ABB RAPID module: KennyTargets.mod

MODULE targets

	!Workplan Variables
	CONST string workplanName := "Kenny";
	CONST string workplanUUID := "4c150834-5da1-4e47-96b7-b16cde8d196c";

	!Workingsteps
	CONST string WorkPlan{20,6} := [
		["1","7", "Drilling.88", "5dba9a8c-05db-4595-a3ca-a7c776a922ef", "Hole.167", "f696efdc-798d-4b52-8da7-1cda0560be94"],
		["8","14", "Drilling.71", "36050cd1-dc9e-4879-8aed-1be84ca47fcc", "Hole.160", "7d9ff765-76db-4167-bb4c-53e49b398220"],
		["15","21", "Drilling.70", "4e2f8e6d-fe62-4a04-8e26-7213540deac3", "Hole.159", "eae91509-0626-466f-8bd8-d981c0f5cb83"],
		["22","28", "Drilling.87", "0659fa42-8109-4895-98a9-1d7bad19a7f8", "Hole.166", "d3306ec8-e7c0-4e48-ab13-ea87fff8c7f5"],
		["29","35", "Drilling.89", "25529f8b-f8c0-4dfe-8d3c-3ee9bb5aaf0b", "Hole.168", "45429ce3-7377-4a4c-ba7a-c1e998d11363"],
		["36","42", "Drilling.72", "0859f91d-f6a2-437f-b292-347030659a13", "Hole.161", "cfed41ef-af78-4deb-868f-e06b5c3e032d"],
		["43","49", "Drilling.87A", "bd213c16-608a-48e8-ba92-16dd103f0e82", "Hole.165", "e244bb89-273f-46de-9470-629b355579d0"],
		["50","56", "Drilling.72A", "30283c33-9bc4-4cb4-8bda-9191e9e1c1a8", "Hole.162", "6466e924-cde5-4cb9-be63-7b2e8a7ccfc9"],
		["57","63", "Drilling.51", "785224d9-9790-4c1a-a5a3-7fdee127c194", "Hole.149", "6ba27eaa-9f1f-4192-92ff-444f81e24c86"],
		["64","70", "Drilling.52", "6f0206cd-ac22-4230-a925-bd17b2c89fdf", "Hole.150", "7cbcafea-7ebf-4eb1-80bd-d38dc37e2ffa"],
		["71","77", "Drilling.52", "8223e776-d7de-4e22-b8f0-fb95f3561672", "Hole.151", "4113edcf-3075-48ef-82ea-78a646f36958"],
		["78","84", "Drilling.53", "15048da7-3430-4dce-a3f8-5c07c276276c", "Hole.152", "8d763157-3777-4192-8350-24f7dbecc6a9"],
		["85","91", "Drilling.66", "95c1f94a-95c9-4216-a369-009bc624fa7c", "Hole.155", "7352fd5f-6f0d-4d28-bb2c-b9767f2ea8ca"],
		["92","98", "Drilling.67", "f632f581-ae96-402c-b4f7-e3bd5086856f", "Hole.156", "7c20ef06-77fc-43ec-8049-9df34a187736"],
		["99","105", "Drilling.68", "c8ae3b54-663b-4d09-baf6-4b0ee80be638", "Hole.157", "0e7d8ffe-7fd5-4dd5-9f70-b0b78f8877dc"],
		["106","112", "Drilling.69", "d220337c-e0a3-4693-a211-54c62b6cd64b", "Hole.158", "6fcc203b-750e-4cab-906d-26d0a8242386"],
		["113","119", "Drilling.90", "f0f7cb38-96f5-48d3-840e-edf378bb551b", "Hole.170", "636bd456-6d68-43b2-b22b-21d689faa8d2"],
		["120","126", "Drilling.91", "abcac725-976e-4a50-a32b-3dd65c42f522", "Hole.171", "d8ca9eb0-5b5f-4eba-8f6d-b2fe1a9acaf1"],
		["127","133", "Drilling.92", "0d36731a-94ab-4213-8ec9-dfebb0effafd", "Hole.172", "f87e6c87-82b4-4795-8769-a91132110e61"],
		["134","140", "Drilling.93", "7777f709-fc7f-49f0-a947-dc19bdc87d5a", "Hole.173", "76d0f419-d37b-4108-8258-5a43c85176e2"]
		];

	!Positions
	CONST robtarget WorkingstepRobtargets{140} := [
		[[1251.36031479439,159.986015149395,27.4616252468863],[0.00827389312568621,0.000714793553765205,-0.996254662433507,0.0860678763663786],[0,0,0,0],[9E+09,9E+09,9E+09,9E+09,9E+09,9E+09]],
		[[1250.52908619628,151.273669125687,-22.5787992695068],[0.00827389312568621,0.000714793553765205,-0.996254662433507,0.0860678763663786],[0,0,0,0],[9E+09,9E+09,9E+09,9E+09,9E+09,9E+09]],
		[[1250.52908619628,151.273669125687,-22.5787992695068],[0.00827389312568621,0.000714793553765205,-0.996254662433507,0.0860678763663786],[0,0,0,0],[9E+09,9E+09,9E+09,9E+09,9E+09,9E+09]],
		[[1250.00956832245,145.828452860869,-53.8540645922525],[0.00827389312568621,0.000714793553765205,-0.996254662433507,0.0860678763663786],[0,0,0,0],[9E+09,9E+09,9E+09,9E+09,9E+09,9E+09]],
		[[1250.00956832245,145.828452860869,-53.8540645922525],[0.00827389312568621,0.000714793553765205,-0.996254662433507,0.0860678763663786],[0,0,0,0],[9E+09,9E+09,9E+09,9E+09,9E+09,9E+09]],
		[[1250.52908619628,151.273669125687,-22.5787992695068],[0.00827389312568621,0.000714793553765205,-0.996254662433507,0.0860678763663786],[0,0,0,0],[9E+09,9E+09,9E+09,9E+09,9E+09,9E+09]],
		[[1251.36031479439,159.986015149395,27.4616252468863],[0.00827389312568621,0.000714793553765205,-0.996254662433507,0.0860678763663786],[0,0,0,0],[9E+09,9E+09,9E+09,9E+09,9E+09,9E+09]],
		[[1190.56655432575,165.147556673713,27.5696380197376],[0.00833481880816476,0.000730999019406425,-0.996141160359995,0.0873658118059379],[0,0,0,0],[9E+09,9E+09,9E+09,9E+09,9E+09,9E+09]],
		[[1189.72949308332,156.304823646231,-22.4478129457116],[0.00833481880816476,0.000730999019406425,-0.996141160359995,0.0873658118059379],[0,0,0,0],[9E+09,9E+09,9E+09,9E+09,9E+09,9E+09]],
		[[1189.72949308332,156.304823646231,-22.4478129457116],[0.00833481880816476,0.000730999019406425,-0.996141160359995,0.0873658118059379],[0,0,0,0],[9E+09,9E+09,9E+09,9E+09,9E+09,9E+09]],
		[[1189.2063298068,150.778115504055,-53.7087197991172],[0.00833481880816476,0.000730999019406425,-0.996141160359995,0.0873658118059379],[0,0,0,0],[9E+09,9E+09,9E+09,9E+09,9E+09,9E+09]],
		[[1189.2063298068,150.778115504055,-53.7087197991172],[0.00833481880816476,0.000730999019406425,-0.996141160359995,0.0873658118059379],[0,0,0,0],[9E+09,9E+09,9E+09,9E+09,9E+09,9E+09]],
		[[1189.72949308332,156.304823646231,-22.4478129457116],[0.00833481880816476,0.000730999019406425,-0.996141160359995,0.0873658118059379],[0,0,0,0],[9E+09,9E+09,9E+09,9E+09,9E+09,9E+09]],
		[[1190.56655432575,165.147556673713,27.5696380197376],[0.00833481880816476,0.000730999019406425,-0.996141160359995,0.0873658118059379],[0,0,0,0],[9E+09,9E+09,9E+09,9E+09,9E+09,9E+09]],
		[[1191.89415560584,213.973804453541,17.5823830985576],[0.00973585929847244,0.00111256490306083,-0.993486175232847,0.113530589993472],[0,0,0,0],[9E+09,9E+09,9E+09,9E+09,9E+09,9E+09]],
		[[1190.92426864878,202.513131068111,-31.8984443484752],[0.00973585929847244,0.00111256490306083,-0.993486175232847,0.113530589993472],[0,0,0,0],[9E+09,9E+09,9E+09,9E+09,9E+09,9E+09]],
		[[1190.92426864878,202.513131068111,-31.8984443484752],[0.00973585929847244,0.00111256490306083,-0.993486175232847,0.113530589993472],[0,0,0,0],[9E+09,9E+09,9E+09,9E+09,9E+09,9E+09]],
		[[1190.31808930061,195.350210202218,-62.8239615028704],[0.00973585929847244,0.00111256490306083,-0.993486175232847,0.113530589993472],[0,0,0,0],[9E+09,9E+09,9E+09,9E+09,9E+09,9E+09]],
		[[1190.31808930061,195.350210202218,-62.8239615028704],[0.00973585929847244,0.00111256490306083,-0.993486175232847,0.113530589993472],[0,0,0,0],[9E+09,9E+09,9E+09,9E+09,9E+09,9E+09]],
		[[1190.92426864878,202.513131068111,-31.8984443484752],[0.00973585929847244,0.00111256490306083,-0.993486175232847,0.113530589993472],[0,0,0,0],[9E+09,9E+09,9E+09,9E+09,9E+09,9E+09]],
		[[1191.89415560584,213.973804453541,17.5823830985576],[0.00973585929847244,0.00111256490306083,-0.993486175232847,0.113530589993472],[0,0,0,0],[9E+09,9E+09,9E+09,9E+09,9E+09,9E+09]],
		[[1251.50868656169,112.759337427171,34.4420178830909],[0.00729205985071979,0.000442363584144468,-0.998138382466358,0.0605508020180991],[0,0,0,0],[9E+09,9E+09,9E+09,9E+09,9E+09,9E+09]],
		[[1250.77191390728,106.618500806138,-15.9800734226999],[0.00729205985071979,0.000442363584144468,-0.998138382466358,0.0605508020180991],[0,0,0,0],[9E+09,9E+09,9E+09,9E+09,9E+09,9E+09]],
		[[1250.77191390728,106.618500806138,-15.9800734226999],[0.00729205985071979,0.000442363584144468,-0.998138382466358,0.0605508020180991],[0,0,0,0],[9E+09,9E+09,9E+09,9E+09,9E+09,9E+09]],
		[[1250.31143099827,102.780477917993,-47.4938804888192],[0.00729205985071979,0.000442363584144468,-0.998138382466358,0.0605508020180991],[0,0,0,0],[9E+09,9E+09,9E+09,9E+09,9E+09,9E+09]],
		[[1250.31143099827,102.780477917993,-47.4938804888192],[0.00729205985071979,0.000442363584144468,-0.998138382466358,0.0605508020180991],[0,0,0,0],[9E+09,9E+09,9E+09,9E+09,9E+09,9E+09]],
		[[1250.77191390728,106.618500806138,-15.9800734226999],[0.00729205985071979,0.000442363584144468,-0.998138382466358,0.0605508020180991],[0,0,0,0],[9E+09,9E+09,9E+09,9E+09,9E+09,9E+09]],
		[[1251.50868656169,112.759337427171,34.4420178830909],[0.00729205985071979,0.000442363584144468,-0.998138382466358,0.0605508020180991],[0,0,0,0],[9E+09,9E+09,9E+09,9E+09,9E+09,9E+09]],
		[[1251.8601825108,210.524561887497,17.2060251950538],[0.0097362625680173,0.00111307904909481,-0.993480782143631,0.113577734426767],[0,0,0,0],[9E+09,9E+09,9E+09,9E+09,9E+09,9E+09]],
		[[1250.89027144533,199.059191507408,-32.2737136338089],[0.0097362625680173,0.00111307904909481,-0.993480782143631,0.113577734426767],[0,0,0,0],[9E+09,9E+09,9E+09,9E+09,9E+09,9E+09]],
		[[1250.89027144533,199.059191507408,-32.2737136338089],[0.0097362625680173,0.00111307904909481,-0.993480782143631,0.113577734426767],[0,0,0,0],[9E+09,9E+09,9E+09,9E+09,9E+09,9E+09]],
		[[1250.28407702942,191.893335019853,-63.1985504018481],[0.0097362625680173,0.00111307904909481,-0.993480782143631,0.113577734426767],[0,0,0,0],[9E+09,9E+09,9E+09,9E+09,9E+09,9E+09]],
		[[1250.28407702942,191.893335019853,-63.1985504018481],[0.0097362625680173,0.00111307904909481,-0.993480782143631,0.113577734426767],[0,0,0,0],[9E+09,9E+09,9E+09,9E+09,9E+09,9E+09]],
		[[1250.89027144533,199.059191507408,-32.2737136338089],[0.0097362625680173,0.00111307904909481,-0.993480782143631,0.113577734426767],[0,0,0,0],[9E+09,9E+09,9E+09,9E+09,9E+09,9E+09]],
		[[1251.8601825108,210.524561887497,17.2060251950538],[0.0097362625680173,0.00111307904909481,-0.993480782143631,0.113577734426767],[0,0,0,0],[9E+09,9E+09,9E+09,9E+09,9E+09,9E+09]],
		[[1190.88023867958,116.257500079554,34.9005826267419],[0.00731948636979851,0.000450203628618277,-0.998086922900926,0.0613898751435108],[0,0,0,0],[9E+09,9E+09,9E+09,9E+09,9E+09,9E+09]],
		[[1190.14080955814,110.031886232754,-15.5110725415314],[0.00731948636979851,0.000450203628618277,-0.998086922900926,0.0613898751435108],[0,0,0,0],[9E+09,9E+09,9E+09,9E+09,9E+09,9E+09]],
		[[1190.14080955814,110.031886232754,-15.5110725415314],[0.00731948636979851,0.000450203628618277,-0.998086922900926,0.0613898751435108],[0,0,0,0],[9E+09,9E+09,9E+09,9E+09,9E+09,9E+09]],
		[[1189.67866635724,106.140877578504,-47.0183570217021],[0.00731948636979851,0.000450203628618277,-0.998086922900926,0.0613898751435108],[0,0,0,0],[9E+09,9E+09,9E+09,9E+09,9E+09,9E+09]],
		[[1189.67866635724,106.140877578504,-47.0183570217021],[0.00731948636979851,0.000450203628618277,-0.998086922900926,0.0613898751435108],[0,0,0,0],[9E+09,9E+09,9E+09,9E+09,9E+09,9E+09]],
		[[1190.14080955814,110.031886232754,-15.5110725415314],[0.00731948636979851,0.000450203628618277,-0.998086922900926,0.0613898751435108],[0,0,0,0],[9E+09,9E+09,9E+09,9E+09,9E+09,9E+09]],
		[[1190.88023867958,116.257500079554,34.9005826267419],[0.00731948636979851,0.000450203628618277,-0.998086922900926,0.0613898751435108],[0,0,0,0],[9E+09,9E+09,9E+09,9E+09,9E+09,9E+09]],
		[[1250.76447640153,68.6402546108708,38.7643104755585],[0.00669120018047459,0.000246507461145111,-0.999299675598547,0.0368147446392719],[0,0,0,0],[9E+09,9E+09,9E+09,9E+09,9E+09,9E+09]],
		[[1250.08604859299,64.9023284513774,-11.8934396100383],[0.00669120018047459,0.000246507461145111,-0.999299675598547,0.0368147446392719],[0,0,0,0],[9E+09,9E+09,9E+09,9E+09,9E+09,9E+09]],
		[[1250.08604859299,64.9023284513774,-11.8934396100383],[0.00669120018047459,0.000246507461145111,-0.999299675598547,0.0368147446392719],[0,0,0,0],[9E+09,9E+09,9E+09,9E+09,9E+09,9E+09]],
		[[1249.66203121265,62.5661246016938,-43.5545334135362],[0.00669120018047459,0.000246507461145111,-0.999299675598547,0.0368147446392719],[0,0,0,0],[9E+09,9E+09,9E+09,9E+09,9E+09,9E+09]],
		[[1249.66203121265,62.5661246016938,-43.5545334135362],[0.00669120018047459,0.000246507461145111,-0.999299675598547,0.0368147446392719],[0,0,0,0],[9E+09,9E+09,9E+09,9E+09,9E+09,9E+09]],
		[[1250.08604859299,64.9023284513774,-11.8934396100383],[0.00669120018047459,0.000246507461145111,-0.999299675598547,0.0368147446392719],[0,0,0,0],[9E+09,9E+09,9E+09,9E+09,9E+09,9E+09]],
		[[1250.76447640153,68.6402546108708,38.7643104755585],[0.00669120018047459,0.000246507461145111,-0.999299675598547,0.0368147446392719],[0,0,0,0],[9E+09,9E+09,9E+09,9E+09,9E+09,9E+09]],
		[[1189.9772715838,69.4582698852428,39.5179868929106],[0.00668793620390687,0.000245146305514718,-0.999306502156587,0.0366295803987568],[0,0,0,0],[9E+09,9E+09,9E+09,9E+09,9E+09,9E+09]],
		[[1189.29916082133,65.7391188387643,-11.1411493145624],[0.00668793620390687,0.000245146305514718,-0.999306502156587,0.0366295803987568],[0,0,0,0],[9E+09,9E+09,9E+09,9E+09,9E+09,9E+09]],
		[[1189.29916082133,65.7391188387643,-11.1411493145624],[0.00668793620390687,0.000245146305514718,-0.999306502156587,0.0366295803987568],[0,0,0,0],[9E+09,9E+09,9E+09,9E+09,9E+09,9E+09]],
		[[1188.87534159478,63.4146494347152,-42.803109444233],[0.00668793620390687,0.000245146305514718,-0.999306502156587,0.0366295803987568],[0,0,0,0],[9E+09,9E+09,9E+09,9E+09,9E+09,9E+09]],
		[[1188.87534159478,63.4146494347152,-42.803109444233],[0.00668793620390687,0.000245146305514718,-0.999306502156587,0.0366295803987568],[0,0,0,0],[9E+09,9E+09,9E+09,9E+09,9E+09,9E+09]],
		[[1189.29916082133,65.7391188387643,-11.1411493145624],[0.00668793620390687,0.000245146305514718,-0.999306502156587,0.0366295803987568],[0,0,0,0],[9E+09,9E+09,9E+09,9E+09,9E+09,9E+09]],
		[[1189.9772715838,69.4582698852428,39.5179868929106],[0.00668793620390687,0.000245146305514718,-0.999306502156587,0.0366295803987568],[0,0,0,0],[9E+09,9E+09,9E+09,9E+09,9E+09,9E+09]],
		[[1048.75377702369,221.064248736861,18.7456359573398],[0.00969862451718228,0.0011013674490227,-0.993566525165611,0.112828559073272],[0,0,0,0],[9E+09,9E+09,9E+09,9E+09,9E+09,9E+09]],
		[[1047.78736158715,209.673531246336,-30.7514103813565],[0.00969862451718228,0.0011013674490227,-0.993566525165611,0.112828559073272],[0,0,0,0],[9E+09,9E+09,9E+09,9E+09,9E+09,9E+09]],
		[[1047.78736158715,209.673531246336,-30.7514103813565],[0.00969862451718228,0.0011013674490227,-0.993566525165611,0.112828559073272],[0,0,0,0],[9E+09,9E+09,9E+09,9E+09,9E+09,9E+09]],
		[[1047.18335193931,202.554332814758,-61.6870643430416],[0.00969862451718228,0.0011013674490227,-0.993566525165611,0.112828559073272],[0,0,0,0],[9E+09,9E+09,9E+09,9E+09,9E+09,9E+09]],
		[[1047.18335193931,202.554332814758,-61.6870643430416],[0.00969862451718228,0.0011013674490227,-0.993566525165611,0.112828559073272],[0,0,0,0],[9E+09,9E+09,9E+09,9E+09,9E+09,9E+09]],
		[[1047.78736158715,209.673531246336,-30.7514103813565],[0.00969862451718228,0.0011013674490227,-0.993566525165611,0.112828559073272],[0,0,0,0],[9E+09,9E+09,9E+09,9E+09,9E+09,9E+09]],
		[[1048.75377702369,221.064248736861,18.7456359573398],[0.00969862451718228,0.0011013674490227,-0.993566525165611,0.112828559073272],[0,0,0,0],[9E+09,9E+09,9E+09,9E+09,9E+09,9E+09]],
		[[1049.72266482233,161.388258470636,30.5369306758237],[0.00810433453815839,0.000668070226723706,-0.996586609691307,0.0821523148051996],[0,0,0,0],[9E+09,9E+09,9E+09,9E+09,9E+09,9E+09]],
		[[1048.90765118534,153.069523657326,-19.5706975246546],[0.00810433453815839,0.000668070226723706,-0.996586609691307,0.0821523148051996],[0,0,0,0],[9E+09,9E+09,9E+09,9E+09,9E+09,9E+09]],
		[[1048.90765118534,153.069523657326,-19.5706975246546],[0.00810433453815839,0.000668070226723706,-0.996586609691307,0.0821523148051996],[0,0,0,0],[9E+09,9E+09,9E+09,9E+09,9E+09,9E+09]],
		[[1048.39826766222,147.870314399008,-50.8879651499535],[0.00810433453815839,0.000668070226723706,-0.996586609691307,0.0821523148051996],[0,0,0,0],[9E+09,9E+09,9E+09,9E+09,9E+09,9E+09]],
		[[1048.39826766222,147.870314399008,-50.8879651499535],[0.00810433453815839,0.000668070226723706,-0.996586609691307,0.0821523148051996],[0,0,0,0],[9E+09,9E+09,9E+09,9E+09,9E+09,9E+09]],
		[[1048.90765118534,153.069523657326,-19.5706975246546],[0.00810433453815839,0.000668070226723706,-0.996586609691307,0.0821523148051996],[0,0,0,0],[9E+09,9E+09,9E+09,9E+09,9E+09,9E+09]],
		[[1049.72266482233,161.388258470636,30.5369306758237],[0.00810433453815839,0.000668070226723706,-0.996586609691307,0.0821523148051996],[0,0,0,0],[9E+09,9E+09,9E+09,9E+09,9E+09,9E+09]],
		[[1050.01208432635,107.933890240474,37.9095374224083],[0.007122245347503,0.00039121136422263,-0.998469455496607,0.0548440244255241],[0,0,0,0],[9E+09,9E+09,9E+09,9E+09,9E+09,9E+09]],
		[[1049.29175162139,102.369982698389,-12.5797094887637],[0.007122245347503,0.00039121136422263,-0.998469455496607,0.0548440244255241],[0,0,0,0],[9E+09,9E+09,9E+09,9E+09,9E+09,9E+09]],
		[[1049.29175162139,102.369982698389,-12.5797094887637],[0.007122245347503,0.00039121136422263,-0.998469455496607,0.0548440244255241],[0,0,0,0],[9E+09,9E+09,9E+09,9E+09,9E+09,9E+09]],
		[[1048.84154368078,98.8925404845857,-44.1354888082459],[0.007122245347503,0.00039121136422263,-0.998469455496607,0.0548440244255241],[0,0,0,0],[9E+09,9E+09,9E+09,9E+09,9E+09,9E+09]],
		[[1048.84154368078,98.8925404845857,-44.1354888082459],[0.007122245347503,0.00039121136422263,-0.998469455496607,0.0548440244255241],[0,0,0,0],[9E+09,9E+09,9E+09,9E+09,9E+09,9E+09]],
		[[1049.29175162139,102.369982698389,-12.5797094887637],[0.007122245347503,0.00039121136422263,-0.998469455496607,0.0548440244255241],[0,0,0,0],[9E+09,9E+09,9E+09,9E+09,9E+09,9E+09]],
		[[1050.01208432635,107.933890240474,37.9095374224083],[0.007122245347503,0.00039121136422263,-0.998469455496607,0.0548440244255241],[0,0,0,0],[9E+09,9E+09,9E+09,9E+09,9E+09,9E+09]],
		[[1048.45280482734,61.188425000286,41.9579660547863],[0.00659046299640987,0.00020471594525679,-0.999496183042603,0.0310468029294715],[0,0,0,0],[9E+09,9E+09,9E+09,9E+09,9E+09,9E+09]],
		[[1047.78419688503,58.0355219643173,-8.73968838666952],[0.00659046299640987,0.00020471594525679,-0.999496183042603,0.0310468029294715],[0,0,0,0],[9E+09,9E+09,9E+09,9E+09,9E+09,9E+09]],
		[[1047.78419688503,58.0355219643173,-8.73968838666952],[0.00659046299640987,0.00020471594525679,-0.999496183042603,0.0310468029294715],[0,0,0,0],[9E+09,9E+09,9E+09,9E+09,9E+09,9E+09]],
		[[1047.36631692108,56.064957566837,-40.4257224125791],[0.00659046299640987,0.00020471594525679,-0.999496183042603,0.0310468029294715],[0,0,0,0],[9E+09,9E+09,9E+09,9E+09,9E+09,9E+09]],
		[[1047.36631692108,56.064957566837,-40.4257224125791],[0.00659046299640987,0.00020471594525679,-0.999496183042603,0.0310468029294715],[0,0,0,0],[9E+09,9E+09,9E+09,9E+09,9E+09,9E+09]],
		[[1047.78419688503,58.0355219643173,-8.73968838666952],[0.00659046299640987,0.00020471594525679,-0.999496183042603,0.0310468029294715],[0,0,0,0],[9E+09,9E+09,9E+09,9E+09,9E+09,9E+09]],
		[[1048.45280482734,61.188425000286,41.9579660547863],[0.00659046299640987,0.00020471594525679,-0.999496183042603,0.0310468029294715],[0,0,0,0],[9E+09,9E+09,9E+09,9E+09,9E+09,9E+09]],
		[[1124.58450857921,76.9515299774283,39.8228669588901],[0.00675250584078808,0.000269433238042634,-0.999182078945179,0.0398685864483636],[0,0,0,0],[9E+09,9E+09,9E+09,9E+09,9E+09,9E+09]],
		[[1123.90010650359,72.904009858962,-10.8110068282249],[0.00675250584078808,0.000269433238042634,-0.999182078945179,0.0398685864483636],[0,0,0,0],[9E+09,9E+09,9E+09,9E+09,9E+09,9E+09]],
		[[1123.90010650359,72.904009858962,-10.8110068282249],[0.00675250584078808,0.000269433238042634,-0.999182078945179,0.0398685864483636],[0,0,0,0],[9E+09,9E+09,9E+09,9E+09,9E+09,9E+09]],
		[[1123.47235520633,70.3743097849206,-42.457177945172],[0.00675250584078808,0.000269433238042634,-0.999182078945179,0.0398685864483636],[0,0,0,0],[9E+09,9E+09,9E+09,9E+09,9E+09,9E+09]],
		[[1123.47235520633,70.3743097849206,-42.457177945172],[0.00675250584078808,0.000269433238042634,-0.999182078945179,0.0398685864483636],[0,0,0,0],[9E+09,9E+09,9E+09,9E+09,9E+09,9E+09]],
		[[1123.90010650359,72.904009858962,-10.8110068282249],[0.00675250584078808,0.000269433238042634,-0.999182078945179,0.0398685864483636],[0,0,0,0],[9E+09,9E+09,9E+09,9E+09,9E+09,9E+09]],
		[[1124.58450857921,76.9515299774283,39.8228669588901],[0.00675250584078808,0.000269433238042634,-0.999182078945179,0.0398685864483636],[0,0,0,0],[9E+09,9E+09,9E+09,9E+09,9E+09,9E+09]],
		[[1126.5993688537,133.371202707924,33.609656791981],[0.00758868592259089,0.000526723182265742,-0.997570999567389,0.0692404161655443],[0,0,0,0],[9E+09,9E+09,9E+09,9E+09,9E+09,9E+09]],
		[[1125.83393655486,126.353057912489,-16.6973979521224],[0.00758868592259089,0.000526723182265742,-0.997570999567389,0.0692404161655443],[0,0,0,0],[9E+09,9E+09,9E+09,9E+09,9E+09,9E+09]],
		[[1125.83393655486,126.353057912489,-16.6973979521224],[0.00758868592259089,0.000526723182265742,-0.997570999567389,0.0692404161655443],[0,0,0,0],[9E+09,9E+09,9E+09,9E+09,9E+09,9E+09]],
		[[1125.35554136809,121.966717415342,-48.139307167187],[0.00758868592259089,0.000526723182265742,-0.997570999567389,0.0692404161655443],[0,0,0,0],[9E+09,9E+09,9E+09,9E+09,9E+09,9E+09]],
		[[1125.35554136809,121.966717415342,-48.139307167187],[0.00758868592259089,0.000526723182265742,-0.997570999567389,0.0692404161655443],[0,0,0,0],[9E+09,9E+09,9E+09,9E+09,9E+09,9E+09]],
		[[1125.83393655486,126.353057912489,-16.6973979521224],[0.00758868592259089,0.000526723182265742,-0.997570999567389,0.0692404161655443],[0,0,0,0],[9E+09,9E+09,9E+09,9E+09,9E+09,9E+09]],
		[[1126.5993688537,133.371202707924,33.609656791981],[0.00758868592259089,0.000526723182265742,-0.997570999567389,0.0692404161655443],[0,0,0,0],[9E+09,9E+09,9E+09,9E+09,9E+09,9E+09]],
		[[1126.0616372464,186.211885781352,24.7464515853499],[0.00880082191675858,0.000856592596021549,-0.995257819874454,0.0968694160272657],[0,0,0,0],[9E+09,9E+09,9E+09,9E+09,9E+09,9E+09]],
		[[1125.18014455072,176.41585939664,-25.0922967706981],[0.00880082191675858,0.000856592596021549,-0.995257819874454,0.0968694160272657],[0,0,0,0],[9E+09,9E+09,9E+09,9E+09,9E+09,9E+09]],
		[[1125.18014455072,176.41585939664,-25.0922967706981],[0.00880082191675858,0.000856592596021549,-0.995257819874454,0.0968694160272657],[0,0,0,0],[9E+09,9E+09,9E+09,9E+09,9E+09,9E+09]],
		[[1124.62921161592,170.293342906194,-56.2415144932284],[0.00880082191675858,0.000856592596021549,-0.995257819874454,0.0968694160272657],[0,0,0,0],[9E+09,9E+09,9E+09,9E+09,9E+09,9E+09]],
		[[1124.62921161592,170.293342906194,-56.2415144932284],[0.00880082191675858,0.000856592596021549,-0.995257819874454,0.0968694160272657],[0,0,0,0],[9E+09,9E+09,9E+09,9E+09,9E+09,9E+09]],
		[[1125.18014455072,176.41585939664,-25.0922967706981],[0.00880082191675858,0.000856592596021549,-0.995257819874454,0.0968694160272657],[0,0,0,0],[9E+09,9E+09,9E+09,9E+09,9E+09,9E+09]],
		[[1126.0616372464,186.211885781352,24.7464515853499],[0.00880082191675858,0.000856592596021549,-0.995257819874454,0.0968694160272657],[0,0,0,0],[9E+09,9E+09,9E+09,9E+09,9E+09,9E+09]],
		[[1124.84625477698,220.957336979353,17.2741397681532],[0.0098367962378513,0.00114012296637116,-0.993301363012953,0.115127493658146],[0,0,0,0],[9E+09,9E+09,9E+09,9E+09,9E+09,9E+09]],
		[[1123.86686698609,209.337597808087,-32.1693882324538],[0.0098367962378513,0.00114012296637116,-0.993301363012953,0.115127493658146],[0,0,0,0],[9E+09,9E+09,9E+09,9E+09,9E+09,9E+09]],
		[[1123.86686698609,209.337597808087,-32.1693882324538],[0.0098367962378513,0.00114012296637116,-0.993301363012953,0.115127493658146],[0,0,0,0],[9E+09,9E+09,9E+09,9E+09,9E+09,9E+09]],
		[[1123.25474961678,202.075260826046,-63.071593232833],[0.0098367962378513,0.00114012296637116,-0.993301363012953,0.115127493658146],[0,0,0,0],[9E+09,9E+09,9E+09,9E+09,9E+09,9E+09]],
		[[1123.25474961678,202.075260826046,-63.071593232833],[0.0098367962378513,0.00114012296637116,-0.993301363012953,0.115127493658146],[0,0,0,0],[9E+09,9E+09,9E+09,9E+09,9E+09,9E+09]],
		[[1123.86686698609,209.337597808087,-32.1693882324538],[0.0098367962378513,0.00114012296637116,-0.993301363012953,0.115127493658146],[0,0,0,0],[9E+09,9E+09,9E+09,9E+09,9E+09,9E+09]],
		[[1124.84625477698,220.957336979353,17.2741397681532],[0.0098367962378513,0.00114012296637116,-0.993301363012953,0.115127493658146],[0,0,0,0],[9E+09,9E+09,9E+09,9E+09,9E+09,9E+09]],
		[[1286.40443376685,208.720093463579,16.9470304734434],[0.00974259835249316,0.00111507411475759,-0.993466087636441,0.113705633560541],[0,0,0,0],[9E+09,9E+09,9E+09,9E+09,9E+09,9E+09]],
		[[1285.43393523947,197.241980312679,-32.5297423710288],[0.00974259835249316,0.00111507411475759,-0.993466087636441,0.113705633560541],[0,0,0,0],[9E+09,9E+09,9E+09,9E+09,9E+09,9E+09]],
		[[1285.43393523947,197.241980312679,-32.5297423710288],[0.00974259835249316,0.00111507411475759,-0.993466087636441,0.113705633560541],[0,0,0,0],[9E+09,9E+09,9E+09,9E+09,9E+09,9E+09]],
		[[1284.82737365986,190.068159593366,-63.4527253988237],[0.00974259835249316,0.00111507411475759,-0.993466087636441,0.113705633560541],[0,0,0,0],[9E+09,9E+09,9E+09,9E+09,9E+09,9E+09]],
		[[1284.82737365986,190.068159593366,-63.4527253988237],[0.00974259835249316,0.00111507411475759,-0.993466087636441,0.113705633560541],[0,0,0,0],[9E+09,9E+09,9E+09,9E+09,9E+09,9E+09]],
		[[1285.43393523947,197.241980312679,-32.5297423710288],[0.00974259835249316,0.00111507411475759,-0.993466087636441,0.113705633560541],[0,0,0,0],[9E+09,9E+09,9E+09,9E+09,9E+09,9E+09]],
		[[1286.40443376685,208.720093463579,16.9470304734434],[0.00974259835249316,0.00111507411475759,-0.993466087636441,0.113705633560541],[0,0,0,0],[9E+09,9E+09,9E+09,9E+09,9E+09,9E+09]],
		[[1286.33124649681,153.926988279123,27.9242514810087],[0.00816312780487694,0.000684952269338226,-0.996464762410529,0.0836114313892439],[0,0,0,0],[9E+09,9E+09,9E+09,9E+09,9E+09,9E+09]],
		[[1285.51062336092,145.461530334075,-22.1587056945564],[0.00816312780487694,0.000684952269338226,-0.996464762410529,0.0836114313892439],[0,0,0,0],[9E+09,9E+09,9E+09,9E+09,9E+09,9E+09]],
		[[1285.51062336092,145.461530334075,-22.1587056945564],[0.00816312780487694,0.000684952269338226,-0.996464762410529,0.0836114313892439],[0,0,0,0],[9E+09,9E+09,9E+09,9E+09,9E+09,9E+09]],
		[[1284.997733901,140.170619118421,-53.4605539292846],[0.00816312780487694,0.000684952269338226,-0.996464762410529,0.0836114313892439],[0,0,0,0],[9E+09,9E+09,9E+09,9E+09,9E+09,9E+09]],
		[[1284.997733901,140.170619118421,-53.4605539292846],[0.00816312780487694,0.000684952269338226,-0.996464762410529,0.0836114313892439],[0,0,0,0],[9E+09,9E+09,9E+09,9E+09,9E+09,9E+09]],
		[[1285.51062336092,145.461530334075,-22.1587056945564],[0.00816312780487694,0.000684952269338226,-0.996464762410529,0.0836114313892439],[0,0,0,0],[9E+09,9E+09,9E+09,9E+09,9E+09,9E+09]],
		[[1286.33124649681,153.926988279123,27.9242514810087],[0.00816312780487694,0.000684952269338226,-0.996464762410529,0.0836114313892439],[0,0,0,0],[9E+09,9E+09,9E+09,9E+09,9E+09,9E+09]],
		[[1280.46270299124,102.38309339464,35.2332574820644],[0.00713645430881742,0.0003960721694737,-0.998437927952443,0.055413158841264],[0,0,0,0],[9E+09,9E+09,9E+09,9E+09,9E+09,9E+09]],
		[[1279.74100171248,96.7616237083952,-15.2495933272039],[0.00713645430881742,0.0003960721694737,-0.998437927952443,0.055413158841264],[0,0,0,0],[9E+09,9E+09,9E+09,9E+09,9E+09,9E+09]],
		[[1279.74100171248,96.7616237083952,-15.2495933272039],[0.00713645430881742,0.0003960721694737,-0.998437927952443,0.055413158841264],[0,0,0,0],[9E+09,9E+09,9E+09,9E+09,9E+09,9E+09]],
		[[1279.28993841325,93.2482051544925,-46.8013750829966],[0.00713645430881742,0.0003960721694737,-0.998437927952443,0.055413158841264],[0,0,0,0],[9E+09,9E+09,9E+09,9E+09,9E+09,9E+09]],
		[[1279.28993841325,93.2482051544925,-46.8013750829966],[0.00713645430881742,0.0003960721694737,-0.998437927952443,0.055413158841264],[0,0,0,0],[9E+09,9E+09,9E+09,9E+09,9E+09,9E+09]],
		[[1279.74100171248,96.7616237083952,-15.2495933272039],[0.00713645430881742,0.0003960721694737,-0.998437927952443,0.055413158841264],[0,0,0,0],[9E+09,9E+09,9E+09,9E+09,9E+09,9E+09]],
		[[1280.46270299124,102.38309339464,35.2332574820644],[0.00713645430881742,0.0003960721694737,-0.998437927952443,0.055413158841264],[0,0,0,0],[9E+09,9E+09,9E+09,9E+09,9E+09,9E+09]],
		[[1279.80555575599,62.0258838013912,38.8434555023548],[0.00663132377542586,0.000222501158844028,-0.999415571315941,0.0335334437457661],[0,0,0,0],[9E+09,9E+09,9E+09,9E+09,9E+09,9E+09]],
		[[1279.13296507583,58.6207271556254,-11.8378283211116],[0.00663132377542586,0.000222501158844028,-0.999415571315941,0.0335334437457661],[0,0,0,0],[9E+09,9E+09,9E+09,9E+09,9E+09,9E+09]],
		[[1279.13296507583,58.6207271556254,-11.8378283211116],[0.00663132377542586,0.000222501158844028,-0.999415571315941,0.0335334437457661],[0,0,0,0],[9E+09,9E+09,9E+09,9E+09,9E+09,9E+09]],
		[[1278.71259590072,56.4925042520218,-43.5136307107779],[0.00663132377542586,0.000222501158844028,-0.999415571315941,0.0335334437457661],[0,0,0,0],[9E+09,9E+09,9E+09,9E+09,9E+09,9E+09]],
		[[1278.71259590072,56.4925042520218,-43.5136307107779],[0.00663132377542586,0.000222501158844028,-0.999415571315941,0.0335334437457661],[0,0,0,0],[9E+09,9E+09,9E+09,9E+09,9E+09,9E+09]],
		[[1279.13296507583,58.6207271556254,-11.8378283211116],[0.00663132377542586,0.000222501158844028,-0.999415571315941,0.0335334437457661],[0,0,0,0],[9E+09,9E+09,9E+09,9E+09,9E+09,9E+09]],
		[[1279.80555575599,62.0258838013912,38.8434555023548],[0.00663132377542586,0.000222501158844028,-0.999415571315941,0.0335334437457661],[0,0,0,0],[9E+09,9E+09,9E+09,9E+09,9E+09,9E+09]]
		];

	!Speeds
	CONST speeddata WorkingstepSpeeddatas{140} := [
		[ 800, 500, 5000, 1000],
		[ 800, 500, 5000, 1000],
		[ 4.23333333333333, 500, 5000, 1000],
		[ 4.23333333333333, 500, 5000, 1000],
		[ 800, 500, 5000, 1000],
		[ 800, 500, 5000, 1000],
		[ 800, 500, 5000, 1000],
		[ 800, 500, 5000, 1000],
		[ 800, 500, 5000, 1000],
		[ 4.23333333333333, 500, 5000, 1000],
		[ 4.23333333333333, 500, 5000, 1000],
		[ 800, 500, 5000, 1000],
		[ 800, 500, 5000, 1000],
		[ 800, 500, 5000, 1000],
		[ 800, 500, 5000, 1000],
		[ 800, 500, 5000, 1000],
		[ 4.23333333333333, 500, 5000, 1000],
		[ 4.23333333333333, 500, 5000, 1000],
		[ 800, 500, 5000, 1000],
		[ 800, 500, 5000, 1000],
		[ 800, 500, 5000, 1000],
		[ 800, 500, 5000, 1000],
		[ 800, 500, 5000, 1000],
		[ 4.23333333333333, 500, 5000, 1000],
		[ 4.23333333333333, 500, 5000, 1000],
		[ 800, 500, 5000, 1000],
		[ 800, 500, 5000, 1000],
		[ 800, 500, 5000, 1000],
		[ 800, 500, 5000, 1000],
		[ 800, 500, 5000, 1000],
		[ 4.23333333333333, 500, 5000, 1000],
		[ 4.23333333333333, 500, 5000, 1000],
		[ 800, 500, 5000, 1000],
		[ 800, 500, 5000, 1000],
		[ 800, 500, 5000, 1000],
		[ 800, 500, 5000, 1000],
		[ 800, 500, 5000, 1000],
		[ 4.23333333333333, 500, 5000, 1000],
		[ 4.23333333333333, 500, 5000, 1000],
		[ 800, 500, 5000, 1000],
		[ 800, 500, 5000, 1000],
		[ 800, 500, 5000, 1000],
		[ 800, 500, 5000, 1000],
		[ 800, 500, 5000, 1000],
		[ 4.23333333333333, 500, 5000, 1000],
		[ 4.23333333333333, 500, 5000, 1000],
		[ 800, 500, 5000, 1000],
		[ 800, 500, 5000, 1000],
		[ 800, 500, 5000, 1000],
		[ 800, 500, 5000, 1000],
		[ 800, 500, 5000, 1000],
		[ 4.23333333333333, 500, 5000, 1000],
		[ 4.23333333333333, 500, 5000, 1000],
		[ 800, 500, 5000, 1000],
		[ 800, 500, 5000, 1000],
		[ 800, 500, 5000, 1000],
		[ 800, 500, 5000, 1000],
		[ 800, 500, 5000, 1000],
		[ 4.23333333333333, 500, 5000, 1000],
		[ 4.23333333333333, 500, 5000, 1000],
		[ 800, 500, 5000, 1000],
		[ 800, 500, 5000, 1000],
		[ 800, 500, 5000, 1000],
		[ 800, 500, 5000, 1000],
		[ 800, 500, 5000, 1000],
		[ 4.23333333333333, 500, 5000, 1000],
		[ 4.23333333333333, 500, 5000, 1000],
		[ 800, 500, 5000, 1000],
		[ 800, 500, 5000, 1000],
		[ 800, 500, 5000, 1000],
		[ 800, 500, 5000, 1000],
		[ 800, 500, 5000, 1000],
		[ 4.23333333333333, 500, 5000, 1000],
		[ 4.23333333333333, 500, 5000, 1000],
		[ 800, 500, 5000, 1000],
		[ 800, 500, 5000, 1000],
		[ 800, 500, 5000, 1000],
		[ 800, 500, 5000, 1000],
		[ 800, 500, 5000, 1000],
		[ 4.23333333333333, 500, 5000, 1000],
		[ 4.23333333333333, 500, 5000, 1000],
		[ 800, 500, 5000, 1000],
		[ 800, 500, 5000, 1000],
		[ 800, 500, 5000, 1000],
		[ 800, 500, 5000, 1000],
		[ 800, 500, 5000, 1000],
		[ 4.23333333333333, 500, 5000, 1000],
		[ 4.23333333333333, 500, 5000, 1000],
		[ 800, 500, 5000, 1000],
		[ 800, 500, 5000, 1000],
		[ 800, 500, 5000, 1000],
		[ 800, 500, 5000, 1000],
		[ 800, 500, 5000, 1000],
		[ 4.23333333333333, 500, 5000, 1000],
		[ 4.23333333333333, 500, 5000, 1000],
		[ 800, 500, 5000, 1000],
		[ 800, 500, 5000, 1000],
		[ 800, 500, 5000, 1000],
		[ 800, 500, 5000, 1000],
		[ 800, 500, 5000, 1000],
		[ 4.23333333333333, 500, 5000, 1000],
		[ 4.23333333333333, 500, 5000, 1000],
		[ 800, 500, 5000, 1000],
		[ 800, 500, 5000, 1000],
		[ 800, 500, 5000, 1000],
		[ 800, 500, 5000, 1000],
		[ 800, 500, 5000, 1000],
		[ 4.23333333333333, 500, 5000, 1000],
		[ 4.23333333333333, 500, 5000, 1000],
		[ 800, 500, 5000, 1000],
		[ 800, 500, 5000, 1000],
		[ 800, 500, 5000, 1000],
		[ 800, 500, 5000, 1000],
		[ 800, 500, 5000, 1000],
		[ 4.23333333333333, 500, 5000, 1000],
		[ 4.23333333333333, 500, 5000, 1000],
		[ 800, 500, 5000, 1000],
		[ 800, 500, 5000, 1000],
		[ 800, 500, 5000, 1000],
		[ 800, 500, 5000, 1000],
		[ 800, 500, 5000, 1000],
		[ 4.23333333333333, 500, 5000, 1000],
		[ 4.23333333333333, 500, 5000, 1000],
		[ 800, 500, 5000, 1000],
		[ 800, 500, 5000, 1000],
		[ 800, 500, 5000, 1000],
		[ 800, 500, 5000, 1000],
		[ 800, 500, 5000, 1000],
		[ 4.23333333333333, 500, 5000, 1000],
		[ 4.23333333333333, 500, 5000, 1000],
		[ 800, 500, 5000, 1000],
		[ 800, 500, 5000, 1000],
		[ 800, 500, 5000, 1000],
		[ 800, 500, 5000, 1000],
		[ 800, 500, 5000, 1000],
		[ 4.23333333333333, 500, 5000, 1000],
		[ 4.23333333333333, 500, 5000, 1000],
		[ 800, 500, 5000, 1000],
		[ 800, 500, 5000, 1000],
		[ 800, 500, 5000, 1000]
		];


ENDMODULE
